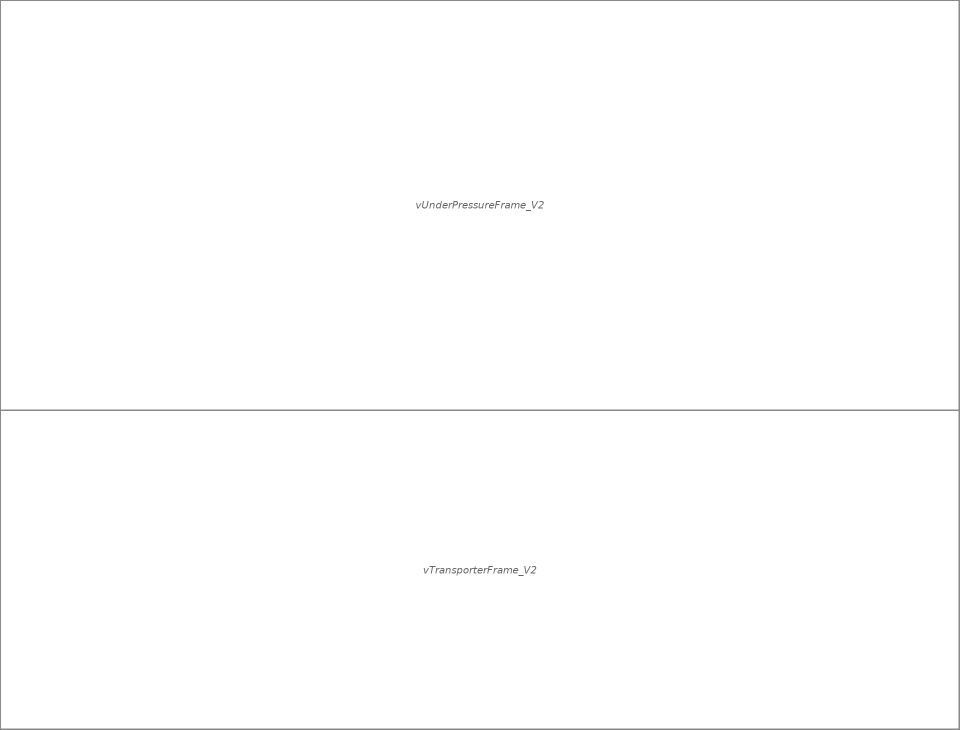
VISUALIZATION vUnderPressureFrame  // 960x730
    Frame (0,410 960x320)
        shows vTransporterFrame_V2(stData := GVL_IO.stTransporterInOuts, stStatus := GVL.stUnderPressureTestStatus, iWorkStep := MAIN.fbTransporterUnderpressure.iWorkStep)
    Frame (0,0 960x410)
        shows vUnderPressureFrame_V2(stInOuts := GVL_IO.stUnderPressureInOuts_V2, stParams := GVL.stUnderPressureTestParams, stStatus := GVL.stUnderPressureTestStatus, iWorkStep := MAIN.fb_UnderPressure_Tester_Machine.iWorkStep)
END_VISUALIZATION

(* stored: Version 1.1.0.1, ProductVersion 3.1.4024.13
   Visu vUnderPressureFrame: Id {6443289e-fcd9-4cc3-a316-39212d567988} *)
